% RSLogix 500 project P10_IVANOVSKI_M.RSS, saved by version 8.30.00.16 %
PROJECT "UNTITLED"    % processor: Bul.1763 MicroLogix 1100 Series B %

PROGRAM FILES
  LAD 2 "MAIN"  5 rungs
  LAD 3 "IO"  11 rungs
  LAD 4 "CONTROLS"  9 rungs
  LAD 5 "ALARMS"  6 rungs

DATA FILES
  O0 OUTPUT  4 elements
  I1 INPUT  6 elements
  S2 STATUS  66 elements
  B3 BINARY  3 elements
  T4 TIMER  4 elements
  C5 COUNTER  1 elements
  R6 CONTROL  1 elements
  N7 INTEGER  5 elements
  F8 FLOAT  1 elements

LADDER 2 "MAIN"
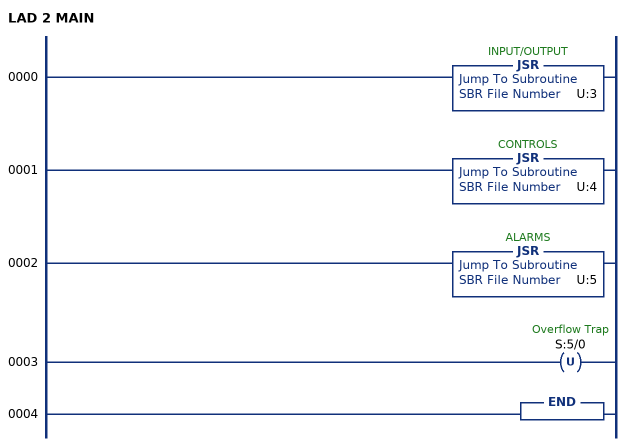
% Rung: 0 %
SOR JSR U:3 EOR
%   U:3  "INPUT/OUTPUT" %
% Rung: 1 %
SOR JSR U:4 EOR
%   U:4  "CONTROLS" %
% Rung: 2 %
SOR JSR U:5 EOR
%   U:5  "ALARMS" %
% Rung: 3 %
SOR OTU S:5/0 EOR
%   S:5/0  "Overflow Trap" %
% Rung: 4 %
SOR END EOR

LADDER 3 "IO"
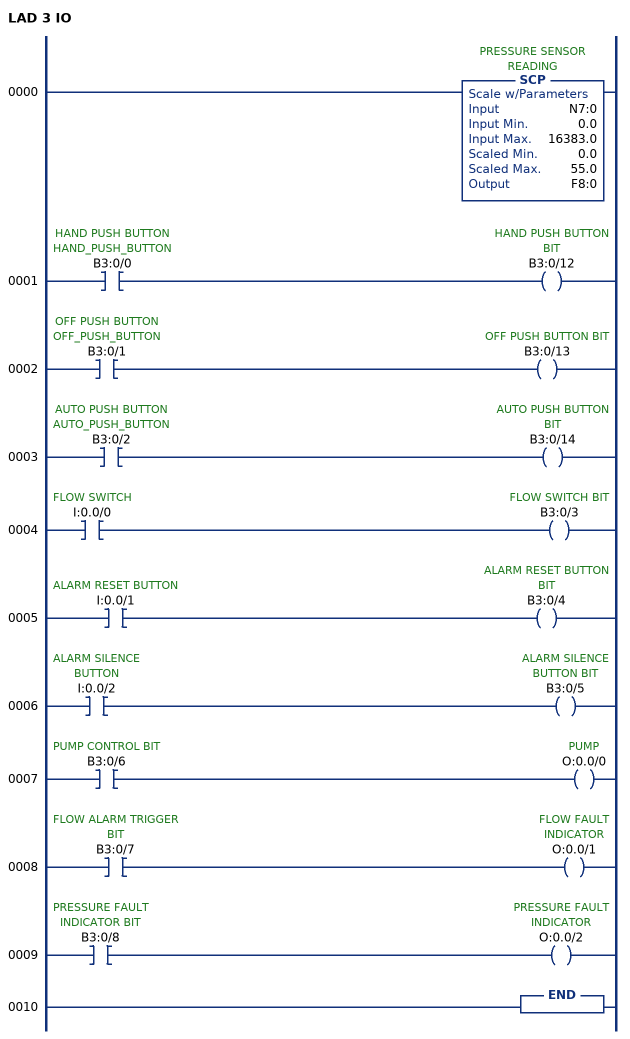
% Rung: 0 %
SOR SCP N7:0 0.0 16383.0 0.0 55.0 F8:0 EOR
%   N7:0  "PRESSURE SENSOR (0-55 PSI)" %
%   F8:0  "PRESSURE SENSOR READING" %
% Rung: 1 %
SOR XIC B3:0/0 OTE B3:0/12 EOR
%   B3:0/0  HAND_PUSH_BUTTON  "HAND PUSH BUTTON" %
%   B3:0/12  "HAND PUSH BUTTON BIT" %
% Rung: 2 %
SOR XIC B3:0/1 OTE B3:0/13 EOR
%   B3:0/1  OFF_PUSH_BUTTON  "OFF PUSH BUTTON" %
%   B3:0/13  "OFF PUSH BUTTON BIT" %
% Rung: 3 %
SOR XIC B3:0/2 OTE B3:0/14 EOR
%   B3:0/2  AUTO_PUSH_BUTTON  "AUTO PUSH BUTTON" %
%   B3:0/14  "AUTO PUSH BUTTON BIT" %
% Rung: 4 %
SOR XIC I:0.0/0 OTE B3:0/3 EOR
%   I:0.0/0  "FLOW SWITCH" %
%   B3:0/3  "FLOW SWITCH BIT" %
% Rung: 5 %
SOR XIC I:0.0/1 OTE B3:0/4 EOR
%   I:0.0/1  "ALARM RESET BUTTON" %
%   B3:0/4  "ALARM RESET BUTTON BIT" %
% Rung: 6 %
SOR XIC I:0.0/2 OTE B3:0/5 EOR
%   I:0.0/2  "ALARM SILENCE BUTTON" %
%   B3:0/5  "ALARM SILENCE BUTTON BIT" %
% Rung: 7 %
SOR XIC B3:0/6 OTE O:0.0/0 EOR
%   B3:0/6  "PUMP CONTROL BIT" %
%   O:0.0/0  "PUMP" %
% Rung: 8 %
SOR XIC B3:0/7 OTE O:0.0/1 EOR
%   B3:0/7  "FLOW ALARM TRIGGER BIT" %
%   O:0.0/1  "FLOW FAULT INDICATOR" %
% Rung: 9 %
SOR XIC B3:0/8 OTE O:0.0/2 EOR
%   B3:0/8  "PRESSURE FAULT INDICATOR BIT" %
%   O:0.0/2  "PRESSURE FAULT INDICATOR" %
% Rung: 10 %
SOR END EOR

LADDER 4 "CONTROLS"
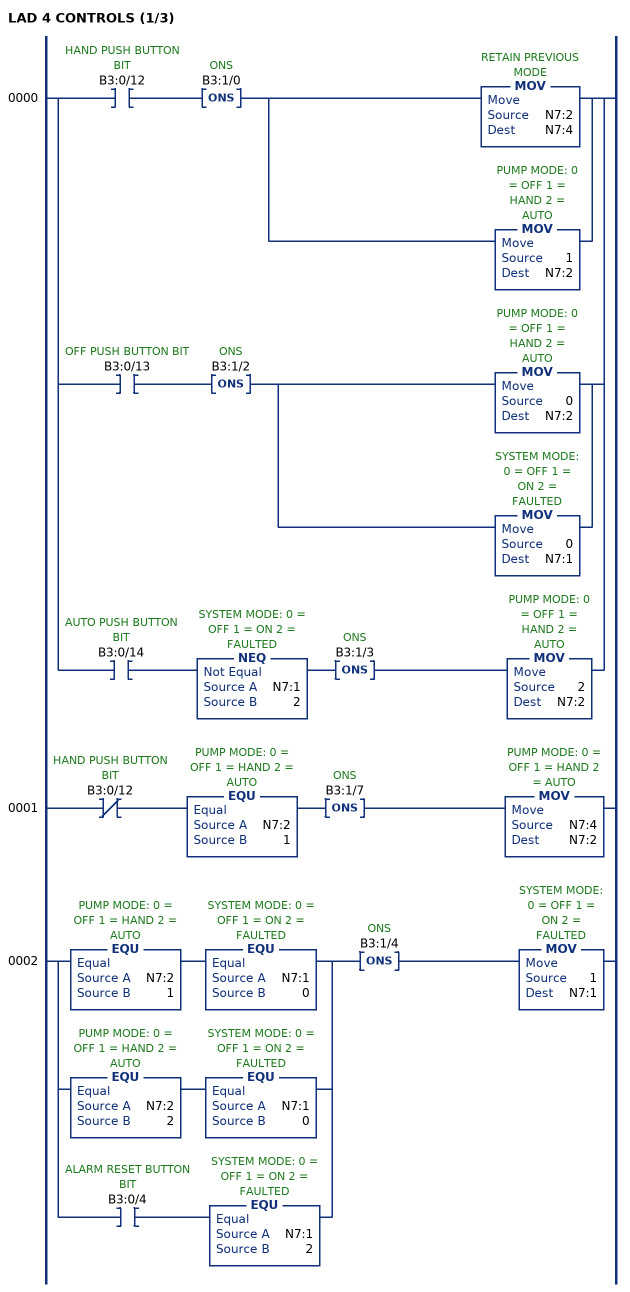
% Rung: 0 %
SOR BST XIC B3:0/12 ONS B3:1/0 BST MOV N7:2 N7:4 NXB MOV 1 N7:2 BND NXB XIC B3:0/13 ONS B3:1/2 BST MOV 0 N7:2 NXB MOV 0 N7:1 BND NXB XIC B3:0/14 NEQ N7:1 2 ONS B3:1/3 MOV 2 N7:2 BND EOR
%   B3:0/12  "HAND PUSH BUTTON BIT" %
%   B3:1/0  "ONS" %
%   N7:2  "PUMP MODE: 0 = OFF 1 = HAND 2 = AUTO" %
%   N7:4  "RETAIN PREVIOUS MODE" %
%   B3:0/13  "OFF PUSH BUTTON BIT" %
%   B3:1/2  "ONS" %
%   N7:1  "SYSTEM MODE: 0 = OFF 1 = ON 2 = FAULTED" %
%   B3:0/14  "AUTO PUSH BUTTON BIT" %
%   B3:1/3  "ONS" %
% Rung: 1 %
SOR XIO B3:0/12 EQU N7:2 1 ONS B3:1/7 MOV N7:4 N7:2 EOR
%   B3:0/12  "HAND PUSH BUTTON BIT" %
%   N7:2  "PUMP MODE: 0 = OFF 1 = HAND 2 = AUTO" %
%   B3:1/7  "ONS" %
%   N7:4  "RETAIN PREVIOUS MODE" %
% Rung: 2 %
SOR BST EQU N7:2 1 EQU N7:1 0 NXB EQU N7:2 2 EQU N7:1 0 NXB XIC B3:0/4 EQU N7:1 2 BND ONS B3:1/4 MOV 1 N7:1 EOR
%   N7:2  "PUMP MODE: 0 = OFF 1 = HAND 2 = AUTO" %
%   N7:1  "SYSTEM MODE: 0 = OFF 1 = ON 2 = FAULTED" %
%   B3:0/4  "ALARM RESET BUTTON BIT" %
%   B3:1/4  "ONS" %

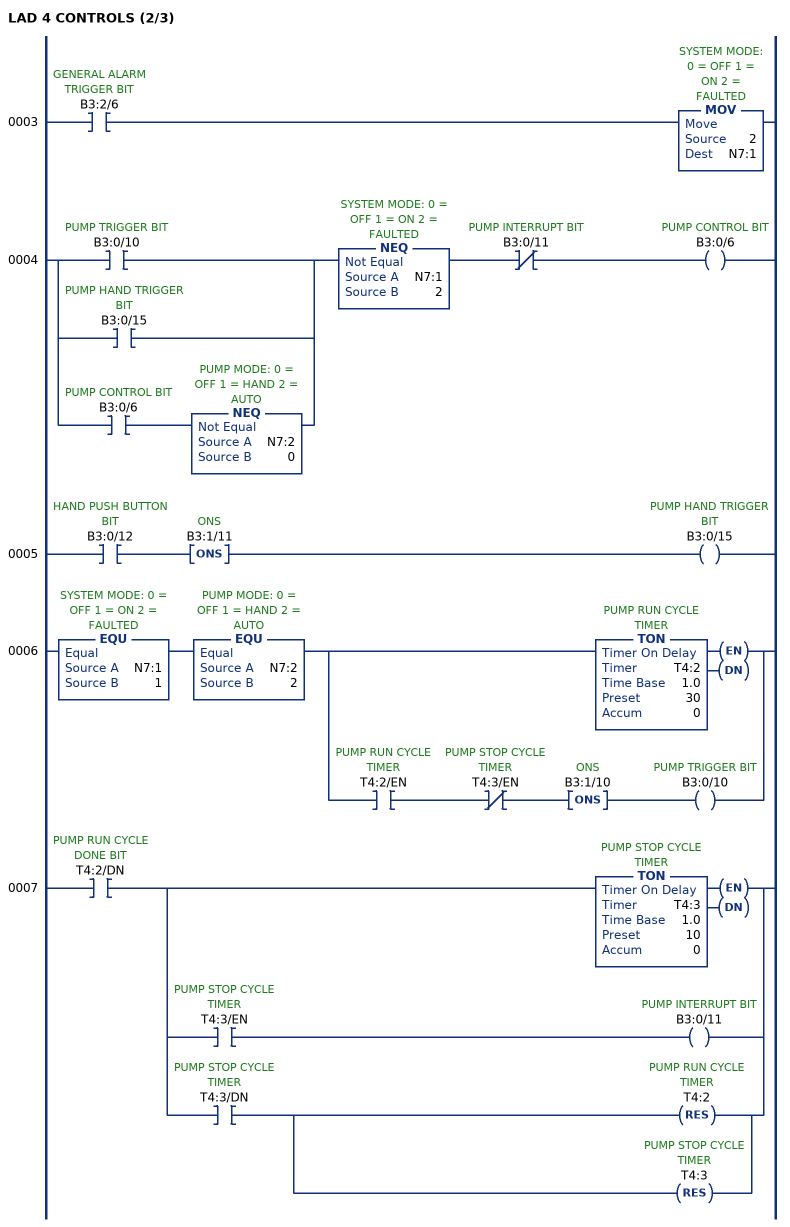
% Rung: 3 %
SOR XIC B3:2/6 MOV 2 N7:1 EOR
%   B3:2/6  "GENERAL ALARM TRIGGER BIT" %
%   N7:1  "SYSTEM MODE: 0 = OFF 1 = ON 2 = FAULTED" %
% Rung: 4 %
SOR BST BST XIC B3:0/10 NXB XIC B3:0/15 BND NXB XIC B3:0/6 NEQ N7:2 0 BND NEQ N7:1 2 XIO B3:0/11 OTE B3:0/6 EOR
%   B3:0/10  "PUMP TRIGGER BIT" %
%   B3:0/15  "PUMP HAND TRIGGER BIT" %
%   B3:0/6  "PUMP CONTROL BIT" %
%   N7:2  "PUMP MODE: 0 = OFF 1 = HAND 2 = AUTO" %
%   N7:1  "SYSTEM MODE: 0 = OFF 1 = ON 2 = FAULTED" %
%   B3:0/11  "PUMP INTERRUPT BIT" %
% Rung: 5 %
SOR XIC B3:0/12 ONS B3:1/11 OTE B3:0/15 EOR
%   B3:0/12  "HAND PUSH BUTTON BIT" %
%   B3:1/11  "ONS" %
%   B3:0/15  "PUMP HAND TRIGGER BIT" %
% Rung: 6 %
SOR EQU N7:1 1 EQU N7:2 2 BST TON T4:2 1.0 30 0 NXB XIC T4:2/EN XIO T4:3/EN ONS B3:1/10 OTE B3:0/10 BND EOR
%   N7:1  "SYSTEM MODE: 0 = OFF 1 = ON 2 = FAULTED" %
%   N7:2  "PUMP MODE: 0 = OFF 1 = HAND 2 = AUTO" %
%   T4:2  "PUMP RUN CYCLE TIMER" %
%   T4:3  "PUMP STOP CYCLE TIMER" %
%   B3:1/10  "ONS" %
%   B3:0/10  "PUMP TRIGGER BIT" %
% Rung: 7 %
SOR XIC T4:2/DN BST TON T4:3 1.0 10 0 NXB XIC T4:3/EN OTE B3:0/11 NXB XIC T4:3/DN BST RES T4:2 NXB RES T4:3 BND BND EOR
%   T4:2/DN  "PUMP RUN CYCLE DONE BIT" %
%   T4:3  "PUMP STOP CYCLE TIMER" %
%   B3:0/11  "PUMP INTERRUPT BIT" %
%   T4:2  "PUMP RUN CYCLE TIMER" %

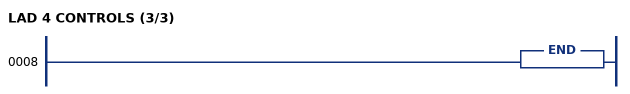
% Rung: 8 %
SOR END EOR

LADDER 5 "ALARMS"
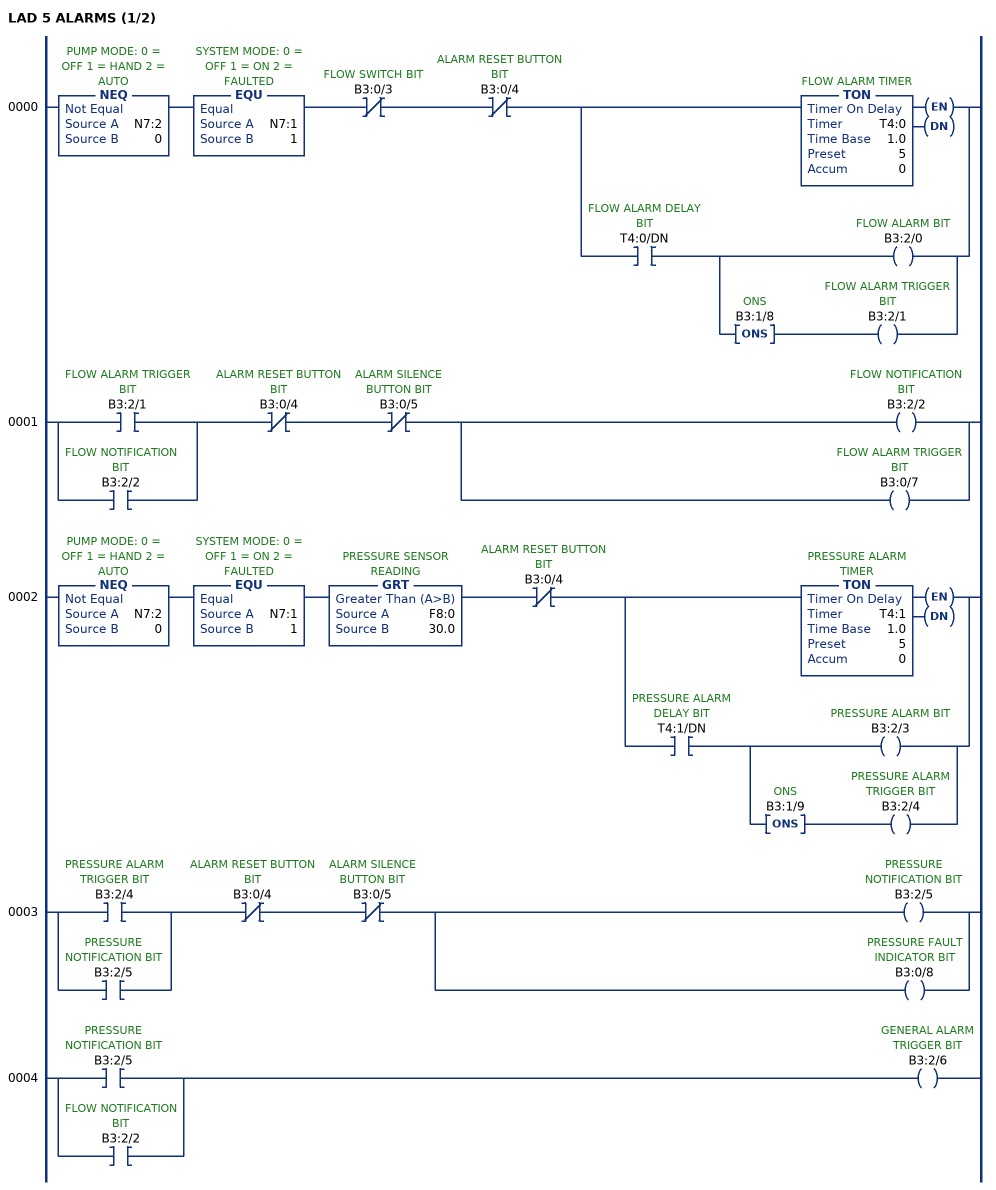
% Rung: 0 %
SOR NEQ N7:2 0 EQU N7:1 1 XIO B3:0/3 XIO B3:0/4 BST TON T4:0 1.0 5 0 NXB XIC T4:0/DN BST OTE B3:2/0 NXB ONS B3:1/8 OTE B3:2/1 BND BND EOR
%   N7:2  "PUMP MODE: 0 = OFF 1 = HAND 2 = AUTO" %
%   N7:1  "SYSTEM MODE: 0 = OFF 1 = ON 2 = FAULTED" %
%   B3:0/3  "FLOW SWITCH BIT" %
%   B3:0/4  "ALARM RESET BUTTON BIT" %
%   T4:0  "FLOW ALARM TIMER" %
%   T4:0/DN  "FLOW ALARM DELAY BIT" %
%   B3:2/0  "FLOW ALARM BIT" %
%   B3:1/8  "ONS" %
%   B3:2/1  "FLOW ALARM TRIGGER BIT" %
% Rung: 1 %
SOR BST XIC B3:2/1 NXB XIC B3:2/2 BND XIO B3:0/4 XIO B3:0/5 BST OTE B3:2/2 NXB OTE B3:0/7 BND EOR
%   B3:2/1  "FLOW ALARM TRIGGER BIT" %
%   B3:2/2  "FLOW NOTIFICATION BIT" %
%   B3:0/4  "ALARM RESET BUTTON BIT" %
%   B3:0/5  "ALARM SILENCE BUTTON BIT" %
%   B3:0/7  "FLOW ALARM TRIGGER BIT" %
% Rung: 2 %
SOR NEQ N7:2 0 EQU N7:1 1 GRT F8:0 30.0 XIO B3:0/4 BST TON T4:1 1.0 5 0 NXB XIC T4:1/DN BST OTE B3:2/3 NXB ONS B3:1/9 OTE B3:2/4 BND BND EOR
%   N7:2  "PUMP MODE: 0 = OFF 1 = HAND 2 = AUTO" %
%   N7:1  "SYSTEM MODE: 0 = OFF 1 = ON 2 = FAULTED" %
%   F8:0  "PRESSURE SENSOR READING" %
%   B3:0/4  "ALARM RESET BUTTON BIT" %
%   T4:1  "PRESSURE ALARM TIMER" %
%   T4:1/DN  "PRESSURE ALARM DELAY BIT" %
%   B3:2/3  "PRESSURE ALARM BIT" %
%   B3:1/9  "ONS" %
%   B3:2/4  "PRESSURE ALARM TRIGGER BIT" %
% Rung: 3 %
SOR BST XIC B3:2/4 NXB XIC B3:2/5 BND XIO B3:0/4 XIO B3:0/5 BST OTE B3:2/5 NXB OTE B3:0/8 BND EOR
%   B3:2/4  "PRESSURE ALARM TRIGGER BIT" %
%   B3:2/5  "PRESSURE NOTIFICATION BIT" %
%   B3:0/4  "ALARM RESET BUTTON BIT" %
%   B3:0/5  "ALARM SILENCE BUTTON BIT" %
%   B3:0/8  "PRESSURE FAULT INDICATOR BIT" %
% Rung: 4 %
SOR BST XIC B3:2/5 NXB XIC B3:2/2 BND OTE B3:2/6 EOR
%   B3:2/5  "PRESSURE NOTIFICATION BIT" %
%   B3:2/2  "FLOW NOTIFICATION BIT" %
%   B3:2/6  "GENERAL ALARM TRIGGER BIT" %

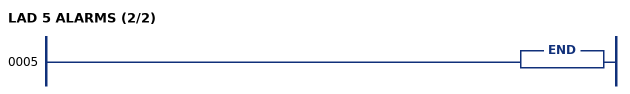
% Rung: 5 %
SOR END EOR

OTHER DOCUMENTED ADDRESSES
  B3:0/9  "FLOW ALARM TRIGGER BIT"
  B3:1/1  "ONS"
  B3:1/5  "ONS"
  B3:1/6  "ONS"
  N7:3  "PRESSURE SENSOR READING"
  U:2  "MAIN"

DATA TABLE (non-zero values as saved)
DATA T4
% .PRE .ACC %
% T4:0 % 5 0
% T4:1 % 5 0
% T4:2 % 30 0
% T4:3 % 10 0
DATA N7
% N7:0 % 8192 0 0 0 0
